(* PLC project FBDexample, Halmstad University FBDexample SNAPSHOT-1.0 *)
(* stored: creationDateTime 2017-08-16T13:43:29, modificationDateTime 2017-08-16T14:46:26 *)

FUNCTION_BLOCK functionBlock1
  VAR
    MPW_AV_S_AcmInhSta_Ewa : BOOL;
    MPW_AV_S_AcmInOpr : BOOL;
    MPW_AV_S_AcmInhSta_Ewb : BOOL;
    MPW_AV_S_AcmInOprRm : BOOL;
    Pt_Sep_CtCl : TIME;
    MPV_AV_C_SepCtCl : BOOL;
    TON0 : TON;
  END_VAR
  VAR  (* added by the conversion: wires and edge detectors of the diagram *)
    _NOT6_OUT : BOOL;
  END_VAR

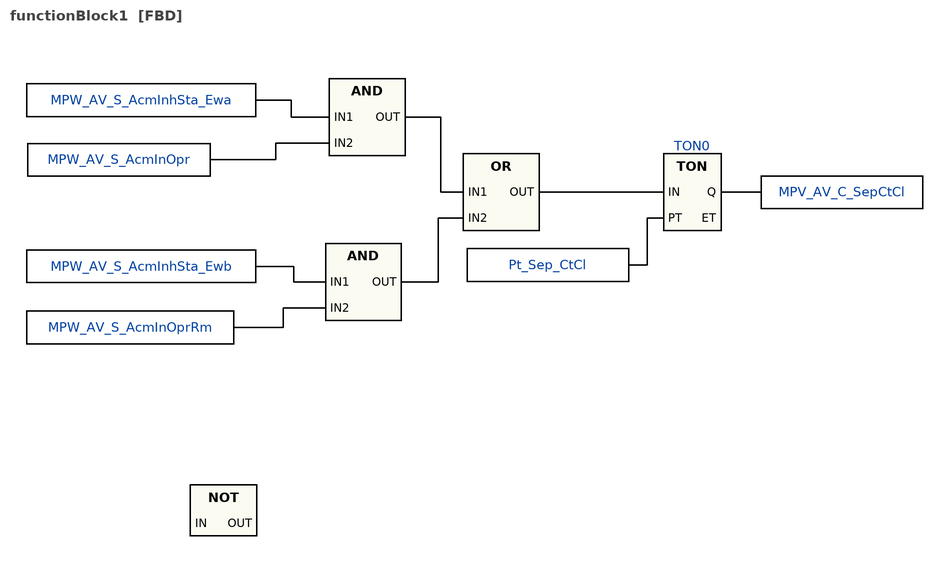
(* FBD diagram, written out as Structured Text *)
TON0(IN := MPW_AV_S_AcmInhSta_Ewa AND MPW_AV_S_AcmInOpr OR MPW_AV_S_AcmInhSta_Ewb AND MPW_AV_S_AcmInOprRm, PT := Pt_Sep_CtCl);
MPV_AV_C_SepCtCl := TON0.Q;
_NOT6_OUT := NOT();
END_FUNCTION_BLOCK
